// TwinCAT 3 PLC project CX7080
// ProgramVersion: 3.1.4024.0
// libraries:
//   Tc2_ControllerToolbox, * (Beckhoff Automation GmbH)
//   Tc2_ModbusRTU, * (Beckhoff Automation GmbH)
//   Tc2_Standard, * (Beckhoff Automation GmbH)
//   Tc2_System, * (Beckhoff Automation GmbH)
//   Tc3_Module, * (Beckhoff Automation GmbH)
// project tree:
//   / PlcTask.TcTTO
//   POUs/ Joint_Control.TcPOU, MAIN.TcPOU, Notes.TcPOU, Notes_Program_funksjonalitet.TcPOU
// real-time tasks:
//   TASK PlcTask: cycle T#10ms, priority 20, ADS port 350
// I/O:
//   DEVICE Device 2 (CX7000), AmsNetId 5.140.122.236.3.1
//   DEVICE Device 4 (COM Port)
// variable links:
//   CX7080/CX7080 Instance <-> Device 4 (COM Port)
//     PlcTask Inputs/MAIN.MB_Master.InData/D[{0..63}] <-> Inputs/Data{1..64}  (64 links)
//     PlcTask Inputs/MAIN.MB_Master.InData/SerStatus <-> Inputs/Status
//     PlcTask Outputs/MAIN.MB_Master.OutData/D[{0..63}] <-> Outputs/Data{1..64}  (64 links)
//     PlcTask Outputs/MAIN.MB_Master.OutData/SerCtrl <-> Outputs/Ctrl

CONFIGURATION CX7080
    RESOURCE PLC ON TwinCAT3
        TASK PlcTask(INTERVAL := T#10ms, PRIORITY := 20);
        PROGRAM MAIN WITH PlcTask : MAIN;
        PROGRAM Joint_Control WITH PlcTask : Joint_Control;
    END_RESOURCE
END_CONFIGURATION

// ---- POUs/MAIN.TcPOU
PROGRAM MAIN
VAR
	MB_Master: ModbusRtuMaster_PcCOM;
	MB_ID: BYTE := 1;
	
	Data_Read : ARRAY[0..9] OF INT;
	Enable_Read: BOOL;
	Busy_Read: BOOL;
	Error_Read : BOOL;
	ErrorId_Read: Tc2_ModbusRTU.MODBUS_ERRORS;
	Register_Read_Address: WORD := 0;

	Data_Write : ARRAY[0..9] OF INT;
	Enable_Write: BOOL;
	Busy_Write: BOOL;
	Error_Write : BOOL;
	ErrorId_Write: Tc2_ModbusRTU.MODBUS_ERRORS;
	Register_Write_Address: WORD := 10;
	
	state : BOOL;
	Toggle_Auto : BOOL := TRUE;
	
	timer: TON;              	// Timer On Delay function block
    clockSignal: BOOL := FALSE; // Output signal that toggles
    period: TIME := T#1MS;  	// Polling frequency
	
	counter : INT;
END_VAR

timer(IN := NOT timer.Q, PT := period);
IF timer.Q THEN
    clockSignal := NOT clockSignal;  // Toggle the signal
END_IF;



MB_Master.ReadRegs(
    UnitID:= MB_ID, 
    Quantity:= 10, 
    MBAddr:= Register_Read_Address, 
    cbLength:= SIZEOF(Data_Read), 
    pMemoryAddr:= ADR(Data_Read), 
    Execute:= Enable_Read, 
    Timeout:= T#100ms, 
    BUSY=> Busy_Read, 
    Error=> Error_Read, 
    ErrorId=> ErrorId_Read, 
    cbRead=>);
	
MB_Master.WriteRegs(
    UnitID:= MB_ID, 
    Quantity:= 10, 
    MBAddr:= Register_Write_Address, 
    cbLength:= SIZEOF(Data_Write), 
    pMemoryAddr:= ADR(Data_Write), 
    Execute:= Enable_Write, 
    Timeout:= T#100ms, 
    BUSY=> Busy_Write, 
    Error=> Error_Write, 
    ErrorId=> ErrorId_Write, 
    cbRead=>);


Data_Write[0] := Joint_Control.Base_Current_Angle;
Data_Write[1] := Joint_Control.Shoulder_Current_Angle;
Data_Write[2] := Joint_Control.Elbow_Current_Angle;
	
IF Toggle_Auto THEN	
	IF clockSignal = TRUE THEN;
		Enable_Read := FALSE;
		Enable_Write := TRUE;
		state := FALSE;
	ELSE
		Enable_Read := TRUE;
		Enable_Write := FALSE;
		state := TRUE;
	END_IF
END_IF;



// Testing

END_PROGRAM

// ---- POUs/Joint_Control.TcPOU
PROGRAM Joint_Control
VAR
	HMI_Base_Angle_Setpoint : INT; 		// [deg] 	Final base angle setpoint from HMI
	HMI_Shoulder_Angle_Setpoint : INT; 	// [deg]	Final shoulder angle setpont from HMI
	HMI_Elbow_Angle_Setpoint : INT; 	// [deg]	Final elbow angle setpoint from HMI
	Base_Current_Angle : INT; 			// [deg]	Intermediate base angle. Calculated in this script with ramp function. Value written to Modbus slave
	Shoulder_Current_Angle : INT; 		// [deg]	Intermediate shoulder angle. Calculated in this script with ramp function. Value written to Modbus slave
	Elbow_Current_Angle : INT; 			// [deg]	Intermediate elbow angle. Calculated in this script with ramp function. Value written to Modbus slave
	HMI_Joint_Ramp_Speed : INT := 10; 	// [deg/s]	Used to set joint speed. Value from HMI
	Ramp_Base : FB_CTRL_RAMP_GENERATOR;
	Ramp_Shoulder : FB_CTRL_RAMP_GENERATOR;
	Ramp_Elbow : FB_CTRL_RAMP_GENERATOR;
	Ramp_Cycle_Time : TIME := T#1ms;
	Ramp_Base_Parameters : ST_CTRL_RAMP_GENERATOR_PARAMS;
	Ramp_Shoulder_Parameters : ST_CTRL_RAMP_GENERATOR_PARAMS;
	Ramp_Elbow_Parameters : ST_CTRL_RAMP_GENERATOR_PARAMS;
END_VAR

IF HMI_Base_Angle_Setpoint > 180 THEN
	HMI_Base_Angle_Setpoint := 180;
ELSIF HMI_Base_Angle_Setpoint < 0 THEN
	HMI_Base_Angle_Setpoint := 0;
END_IF

IF HMI_Shoulder_Angle_Setpoint > 180 THEN
	HMI_Shoulder_Angle_Setpoint := 180;
ELSIF HMI_Shoulder_Angle_Setpoint < 0 THEN
	HMI_Shoulder_Angle_Setpoint := 0;
END_IF

IF HMI_Elbow_Angle_Setpoint > 180 THEN
	HMI_Elbow_Angle_Setpoint := 180;
ELSIF HMI_Elbow_Angle_Setpoint < 0 THEN
	HMI_Elbow_Angle_Setpoint := 0;
END_IF


Ramp_Base_Parameters.fVeloNeg := HMI_Joint_Ramp_Speed;
Ramp_Base_Parameters.fVeloPos := HMI_Joint_Ramp_Speed;
Ramp_Base_Parameters.tCtrlCycleTime := Ramp_Cycle_Time;
Ramp_Base_Parameters.tTaskCycleTime := Ramp_Cycle_Time;
Ramp_Base.bEnable := TRUE;
Ramp_Base(stParams := Ramp_Base_Parameters);


Ramp_Shoulder_Parameters.fVeloNeg := HMI_Joint_Ramp_Speed;
Ramp_Shoulder_Parameters.fVeloPos := HMI_Joint_Ramp_Speed;
Ramp_Shoulder_Parameters.tCtrlCycleTime := Ramp_Cycle_Time;
Ramp_Shoulder_Parameters.tTaskCycleTime := Ramp_Cycle_Time;
Ramp_Shoulder.bEnable := TRUE;
Ramp_Shoulder(stParams := Ramp_Shoulder_Parameters);


Ramp_Elbow_Parameters.fVeloNeg := HMI_Joint_Ramp_Speed;
Ramp_Elbow_Parameters.fVeloPos := HMI_Joint_Ramp_Speed;
Ramp_Elbow_Parameters.tCtrlCycleTime := Ramp_Cycle_Time;
Ramp_Elbow_Parameters.tTaskCycleTime := Ramp_Cycle_Time;
Ramp_Elbow.bEnable := TRUE;
Ramp_Elbow(stParams := Ramp_Elbow_Parameters);


Ramp_Base.fStart := HMI_Base_Angle_Setpoint;
Ramp_Shoulder.fStart := HMI_Shoulder_Angle_Setpoint;
Ramp_Elbow.fStart := HMI_Elbow_Angle_Setpoint;

Ramp_Base.fTarget := HMI_Base_Angle_Setpoint;
Ramp_Shoulder.fTarget := HMI_Shoulder_Angle_Setpoint;
Ramp_Elbow.fTarget := HMI_Elbow_Angle_Setpoint;

Base_Current_Angle := LREAL_TO_INT(Ramp_Base.fOut);
Shoulder_Current_Angle := LREAL_TO_INT(Ramp_Shoulder.fOut);
Elbow_Current_Angle := LREAL_TO_INT(Ramp_Elbow.fOut);

END_PROGRAM

// ---- POUs/Notes.TcPOU
PROGRAM Notes
VAR
END_VAR

(*
Har implementert følgende:
- Modbus RTU read og write registers program
- Versjonskontroll/Git
- Har opprettet HMI prosjekt for å vise register verdier
- Spesifisere hva dette programmet skal kunne gjøre
- Sjekke om det finnes allerede eksisterende blokker som har funksjonaliteten jeg ønsker
- Spesifiser hvordan HMI skal se ut

Videre oppgaver:
- Prøve å gå tilbake til en eldre versjon ved hjelp av Git. Lag eget prosjekt for dette
- Implementere bibliotek for testing av funksjonsblokker/TcUnit
- Lage eget bibliotek for egne implementerte funksjonsblokker som er testet med TcUnit




*)

END_PROGRAM

// ---- POUs/Notes_Program_funksjonalitet.TcPOU
PROGRAM Notes_Program_funksjonalitet
VAR
END_VAR

(*
- Skal kunne manuelt "jogge roboten dit man vil ved hjelp knapper på skjermen"
- Skal kunne lagre koordinater som roboten skal bevege seg mellom
- Skal kunne justere hastigheten som roboten beveger seg mellom 10 og 100% hastighet
- Skal bruke "scope" funksjonen for å plotte ønskede vinkler mot nåværende vinkler
*)

END_PROGRAM
